(* LS Electric XG5000 project: SureServo2_FB *)
(* PLC LSPLC *)
(* module base 0 slot 0: Input/Output Module:XEM-DN/DP32HP (DC 24V Input, Transistor Output, 32 Contacts) *)
(* module base 0 slot 1: Internal Positioning:XBF-PO06E (Open Collector Type, 6 Axis) *)
(* module base 0 slot 2: EtherNet/IP:XBL-EIPT (EtherNet/IP communication module, electrical) *)
VAR_GLOBAL
    SureServo2_EIP_Input00 : ARRAY[0..63] OF BYTE; (* Input data to Ethernet/IP SureServo2 drive *)
    SureServo2_EIP_Output00 : ARRAY[0..63] OF BYTE; (* Output data to Ethernet/IP SureServo2 drive *)
END_VAR

(* Comments on direct variables
%IX0.0.0	this is comment 1
*)

TYPE SureServo2_EIP_UDT : (* Data type for accessing inputs and outputs of a Nitra PAL EIP manifold. *)
STRUCT
    Status_Z_Phase_Offset : DINT; (* z phase offset of Sure servo 2 *)
    Status_Position_Feedback : DINT; (* current position *)
    Status_Speed_Feedback : DINT; (* current speed *)
    Status_Torque_Feedback : DINT; (* current torque *)
    Integrated_DI_Status : DWORD; (* integrated digital inputs *)
    Status_Servo_Alarm : INT; (* current servo alarm *)
    Status_Path_Target_Status : INT; (* status of path target command.  servo should be in PR control mode. *)
    Status_Servo_Ready : BOOL; (* Servo is ready for commands *)
    Status_Servo_Enabled : BOOL; (* Servo has been enabled *)
    Status_Zero_Speed : BOOL; (* Servo is at zero speed *)
    Status_Target_Speed_Reached : BOOL; (* target speed has been reached *)
    Status_Target_Position_Reached : BOOL; (* target position has been reached *)
    Status_Torque_Limit_Reached : BOOL; (* torque limit has been reached. *)
    Status_Alarm : BOOL; (* drive alarm status *)
    Status_Brake_On : BOOL; (* motor brake status *)
    Status_Home : BOOL; (* axis is at home. *)
    Status_Motor_Overload : BOOL; (* status that the motor is overloaded *)
    Status_Warning : BOOL; (* status that there is a drive warning. *)
    Control_Speed_CMD3 : DINT; (* speed command *)
    Control_Servo_Enable : BOOL; (* command to enable the servo *)
    Control_Alarm_Reset : BOOL; (* command to reset an alarm *)
    Control_Speed_PR_Mode : BOOL; (* command for speed or path target mode *)
    Control_Trigger : BOOL; (* trigger command *)
    Control_PR_Select_0 : BOOL; (* path target mode 0 *)
    Control_Stop : BOOL; (* Stop motion command *)
    Control_EStop : BOOL; (* emergency stop status *)
    Control_ECAM_On : BOOL; (* command to turn on ECAM functionality *)
    Control_PR_Path_Target : UINT; (* Path target value *)
    Control_PR_Path_Trigger : UINT; (* Path target trigger value. *)
END_STRUCT;
END_TYPE

FUNCTION_BLOCK SureServo2_EIP_FB
(* function block for SureServo2 parameters over EtherNet/IP *)
VAR_INPUT
    Enable : BOOL; (* Enable the FB. *)
    Source_InputData : ARRAY[0..63] OF BYTE; (* This is the input data from EIP Block of Nitra PAL in the P2P settings. *)
END_VAR
VAR_IN_OUT
    Source_OutputData : ARRAY[0..63] OF BYTE; (* This is the output data from EIP Block of Nitra PAL in the P2P settings. *)
    User_UDT : SureServo2_EIP_UDT; (* This is user declared udt for the SureServo2 EIP FB *)
END_VAR
VAR_OUTPUT
    Active : BOOL; (* status that function block is enabled. *)
END_VAR
VAR
    Destination_OutputData : ARRAY[0..63] OF BYTE; (* Data to be copied into Source_OutputData after every loop. *)
    IP0010_Monitoring_Parameter : DWORD; (* temporary dword storage for input parameter 00.10 *)
    IP0011_Monitoring_Parameter : DWORD; (* temporary dword storage for input parameter 00.11 *)
    IP0012_Monitoring_Parameter : DWORD; (* temporary dword storage for input parameter 00.12 *)
    IP0013_Monitoring_Parameter : DWORD; (* temporary dword storage for input parameter 00.13 *)
    IP0025_Monitoring_Parameter : DWORD; (* temporary dword storage for input parameter 00.25 *)
    IP0026_Monitoring_Parameter : DWORD; (* temporary dword storage for input parameter 00.26 *)
    IP009_Monitoring_Parameter : DWORD; (* temporary dword storage for input parameter 00.09 *)
    OP0029_Mapping_Parameter : DWORD; (* temporary dword storage for output parameter 00.29 *)
    OP0030_Mapping_Parameter : DWORD; (* temporary dword storage for output parameter 00.30 *)
    OP0032_Mapping_Parameter : DWORD; (* temporary dword storage for output parameter 00.32 *)
    TempWord1 : WORD; (* temporary word storage *)
    TempWord2 : WORD; (* temporary word storage *)
END_VAR
(* 
AutomationDirect.com has provided this code for convenience. This sample code is provided "as-is" with no expressed or implied warranty. 
 If the end user includes any of the sample code (in whole or part), it is the user's responsibility to completely modify, integrate, and test any code to ensure it meets all system and 
 safety requirements for the intended application or system.
 *)

(* Only run function block if enable is true *)
IF (Enable = TRUE) THEN
		Active := TRUE;
		
		(*Create DWORDS of input data.  Helps split it up according to SS2 parameters *)
		TempWord1 := BYTE_WORD(LOW:=Source_InputData[0], HIGH:=Source_InputData[1]);
		TempWord2 := BYTE_WORD(LOW:=Source_InputData[2], HIGH:=Source_InputData[3]);		
		IP009_Monitoring_Parameter :=WORD_DWORD(LOW:=TempWord1, HIGH:=TempWord2);
		
		TempWord1 := BYTE_WORD(LOW:=Source_InputData[4], HIGH:=Source_InputData[5]);
		TempWord2 := BYTE_WORD(LOW:=Source_InputData[6], HIGH:=Source_InputData[7]);	
		IP0010_Monitoring_Parameter :=WORD_DWORD(LOW:=TempWord1, HIGH:=TempWord2);
		
		TempWord1 := BYTE_WORD(LOW:=Source_InputData[8], HIGH:=Source_InputData[9]);
		TempWord2 := BYTE_WORD(LOW:=Source_InputData[10], HIGH:=Source_InputData[11]);	
		IP0011_Monitoring_Parameter :=WORD_DWORD(LOW:=TempWord1, HIGH:=TempWord2);
		
		TempWord1 := BYTE_WORD(LOW:=Source_InputData[12], HIGH:=Source_InputData[13]);
		TempWord2 := BYTE_WORD(LOW:=Source_InputData[14], HIGH:=Source_InputData[15]);	
		IP0012_Monitoring_Parameter :=WORD_DWORD(LOW:=TempWord1, HIGH:=TempWord2);
		
		TempWord1 := BYTE_WORD(LOW:=Source_InputData[16], HIGH:=Source_InputData[17]);
		TempWord2 := BYTE_WORD(LOW:=Source_InputData[18], HIGH:=Source_InputData[19]);	
		IP0013_Monitoring_Parameter :=WORD_DWORD(LOW:=TempWord1, HIGH:=TempWord2);
		
		(*
		TempWord1 := BYTE_WORD(LOW:=Source_InputData[20], HIGH:=Source_InputData[21]);
		TempWord2 := BYTE_WORD(LOW:=Source_InputData[22], HIGH:=Source_InputData[23]);	
		IP0025_Monitoring_Parameter :=WORD_DWORD(LOW:=TempWord1, HIGH:=TempWord2);
		
		TempWord1 := BYTE_WORD(LOW:=Source_InputData[24], HIGH:=Source_InputData[25]);
		TempWord2 := BYTE_WORD(LOW:=Source_InputData[26], HIGH:=Source_InputData[27]);	
		IP0026_Monitoring_Parameter :=WORD_DWORD(LOW:=TempWord1, HIGH:=TempWord2);  *)
		 
		
		(* Map Inputs from SS2 Drive *)
		TempWord1 := BYTE_WORD(LOW:=Source_InputData[20], HIGH:=Source_InputData[21]);
		User_UDT.Status_Servo_Ready := TempWord1.0;
		User_UDT.Status_Servo_Enabled := TempWord1.1;
		User_UDT.Status_Zero_Speed := TempWord1.2;
		User_UDT.Status_Target_Speed_Reached := TempWord1.3;
		User_UDT.Status_Target_Position_Reached := TempWord1.4;
		User_UDT.Status_Torque_Limit_Reached := TempWord1.5;
		User_UDT.Status_Alarm := TempWord1.6;
		User_UDT.Status_Brake_On := TempWord1.7;
		User_UDT.Status_Home := TempWord1.8;
		User_UDT.Status_Motor_Overload := TempWord1.9;
		User_UDT.Status_Warning := TempWord1.10;
		
		
		User_UDT.Status_Z_Phase_Offset := DWORD_TO_DINT(IP009_Monitoring_Parameter);
		User_UDT.Status_Position_Feedback := DWORD_TO_DINT(IP0010_Monitoring_Parameter);
		User_UDT.Status_Speed_Feedback := DWORD_TO_DINT(IP0011_Monitoring_Parameter);
		User_UDT.Status_Torque_Feedback := DWORD_TO_DINT(IP0012_Monitoring_Parameter);
		User_UDT.Integrated_DI_Status := IP0013_Monitoring_Parameter;
		
		TempWord2 := BYTE_WORD(LOW:=Source_InputData[22], HIGH:=Source_InputData[23]);	
		User_UDT.Status_Servo_Alarm := WORD_TO_INT(IN:=TempWord2);
		
		TempWord1 := BYTE_WORD(LOW:=Source_InputData[24], HIGH:=Source_InputData[25]);
		User_UDT.Status_Path_Target_Status := WORD_TO_INT(IN:=TempWord1);
		
	
	
		(* Map Outputs to SS2 Drive *)
		OP0029_Mapping_Parameter.0 := User_UDT.Control_Servo_Enable;
		OP0029_Mapping_Parameter.1 := User_UDT.Control_Alarm_Reset;
		OP0029_Mapping_Parameter.2 := User_UDT.Control_Speed_PR_Mode;
		OP0029_Mapping_Parameter.3 := User_UDT.Control_Trigger;
		OP0029_Mapping_Parameter.4 := User_UDT.Control_PR_Select_0;
		OP0029_Mapping_Parameter.5 := User_UDT.Control_Stop;
		OP0029_Mapping_Parameter.6 := User_UDT.Control_EStop;
		OP0029_Mapping_Parameter.7 := User_UDT.Control_ECAM_On;
		
		TempWord1 := UINT_TO_WORD(IN:=User_UDT.Control_PR_Path_Target);
		TempWord2 := UINT_TO_WORD(IN:=User_UDT.Control_PR_Path_Trigger);		
		OP0030_Mapping_Parameter := WORD_DWORD(LOW:=TempWord1, HIGH:=TempWord2);
		
		OP0032_Mapping_Parameter := DINT_TO_DWORD(User_UDT.Control_Speed_CMD3);
	
		//convert DWORD data to bytes for source output data	
		DWORD_WORD(IN:=OP0029_Mapping_Parameter, LOW=>TempWord1, HIGH=>TempWord2);
		WORD_BYTE(IN:=TempWord1, LOW=>Destination_OutputData	[0], HIGH=>Destination_OutputData[1]);
		WORD_BYTE(IN:=TempWord2, LOW=>Destination_OutputData[2], HIGH=>Destination_OutputData[3]);
		 
		DWORD_WORD(IN:=OP0030_Mapping_Parameter, LOW=>TempWord1, HIGH=>TempWord2);
		WORD_BYTE(IN:=TempWord1, LOW=>Destination_OutputData	[4], HIGH=>Destination_OutputData[5]);
		WORD_BYTE(IN:=TempWord2, LOW=>Destination_OutputData[6], HIGH=>Destination_OutputData[7]);
		
		DWORD_WORD(IN:=OP0032_Mapping_Parameter, LOW=>TempWord1, HIGH=>TempWord2);
		WORD_BYTE(IN:=TempWord1, LOW=>Destination_OutputData	[12], HIGH=>Destination_OutputData[13]);
		WORD_BYTE(IN:=TempWord2, LOW=>Destination_OutputData[14], HIGH=>Destination_OutputData[15]);
		 
	
		(* Copy temporary output data array to the source output that gets sent to the PAL unit *)
		Source_OutputData := ARY_MOVE(MOVE_NUM:= 64, IN:=Destination_OutputData, IN_INDX:=0, OUT_INDX:=0);

ELSE	
	Active := FALSE;
	
END_IF; //end of enable if
END_FUNCTION_BLOCK

PROGRAM FB_Usage_LD (* task: Scan Program *)
VAR
    SS2_Drive_Control00 : SureServo2_EIP_UDT; (* User data type for sure servo 2 fb. *)
    SS2_Drive_FB00 : SureServo2_EIP_FB; (* function block instance for sure servo 2 *)
END_VAR
VAR_EXTERNAL
    SureServo2_EIP_Input00 : ARRAY[0..63] OF BYTE; (* Input data to Ethernet/IP SureServo2 drive *)
    SureServo2_EIP_Output00 : ARRAY[0..63] OF BYTE; (* Output data to Ethernet/IP SureServo2 drive *)
END_VAR

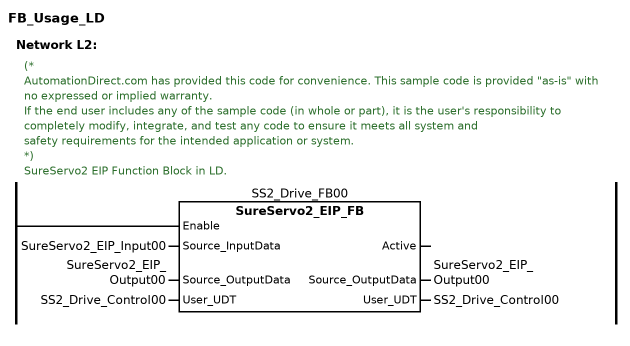
(* ( * / AutomationDirect.com has provided this code for convenience. This sample code is provided "as-is" with no expressed or implied warranty. / If the end user includes any of the sample code (in whole or part), it is the user's responsibility to completely modify, integrate, and test any code to ensure it meets all system and / safety requirements for the intended application or system. / * ) *)
(* SureServo2 EIP Function Block in LD. *)
(* Rung L2 *)
SS2_Drive_FB00(Enable := TRUE, Source_InputData := SureServo2_EIP_Input00, Source_OutputData := SureServo2_EIP_Output00, User_UDT := SS2_Drive_Control00, Source_OutputData => SureServo2_EIP_Output00, User_UDT => SS2_Drive_Control00);
END_PROGRAM

PROGRAM FB_Usage_ST (* task: Scan Program *)
(*  *)
VAR
    fbActive : BOOL; (* local variable for function block active status *)
    SS2_Drive_Control00 : SureServo2_EIP_UDT; (* User data type for sure servo 2 fb. *)
    SS2_FB00 : SureServo2_EIP_FB; (* function block instance for sure servo 2 *)
END_VAR
VAR_EXTERNAL
    SureServo2_EIP_Input00 : ARRAY[0..63] OF BYTE; (* Input data to Ethernet/IP SureServo2 drive *)
    SureServo2_EIP_Output00 : ARRAY[0..63] OF BYTE; (* Output data to Ethernet/IP SureServo2 drive *)
END_VAR
(* 
AutomationDirect.com has provided this code for convenience. This sample code is provided "as-is" with no expressed or implied warranty. 
 If the end user includes any of the sample code (in whole or part), it is the user's responsibility to completely modify, integrate, and test any code to ensure it meets all system and 
 safety requirements for the intended application or system.
 *)


SS2_FB00(Enable:=TRUE, Source_InputData:=SureServo2_EIP_Input00, Source_OutputData:=SureServo2_EIP_Output00, User_UDT:=SS2_Drive_Control00, Active=>fbActive);
END_PROGRAM